Yaskawa INFORM job: X2_242(90,180)_HARDOX.JBI

/JOB
//NAME X2_242(90,180)_HARDOX
///FOLDERNAME X2
//POS
///NPOS 237,237,237,7,0,0
///TOOL 0
///POSTYPE PULSE
///PULSE
C00000=2000,-130321,-133031,0,28968,0
C00001=117091,-130321,-133031,-2123,28968,3391
C00002=159919,-130321,-133031,-2123,28968,3391
C00003=159919,-130321,-133031,-2123,87939,3391
C00004=105022,-108859,-78959,31083,72176,68730
C00005=151007,-25092,-39063,12800,65605,-78235
C00006=132593,67036,12002,14068,96381,-18620
C00007=133669,66493,21901,13656,90017,-18991
C00008=134323,89636,48442,14320,95130,-18049
C00009=134323,89198,49863,14289,94064,-18173
C00010=134090,67791,24612,13544,88977,-18967
C00011=134777,68740,27409,13371,87669,-18883
C00012=134996,69719,28564,13316,87433,-18835
C00013=134996,70471,26931,13315,88788,-18690
C00014=132576,62954,16151,13952,91863,-19138
C00015=158058,56370,5063,6789,93126,12165
C00016=161492,61731,13256,13118,78465,26852
C00017=161219,65846,21027,13360,75906,26484
C00018=158063,89381,46849,19528,82253,27212
C00019=158063,88948,47996,19566,81373,27071
C00020=160512,68550,26920,13794,73840,26014
C00021=160268,69078,27542,13908,73773,25920
C00022=161163,66904,24770,13484,74201,26276
C00023=161204,69435,27921,13504,73574,26218
C00024=161316,71640,30535,13487,73093,26202
C00025=161111,67594,24408,13472,74770,26322
C00026=161490,61134,14077,13154,77673,26766
C00027=158729,69794,18853,21227,92144,29458
C00028=158729,68570,20268,21195,90741,29212
C00029=158729,67854,21249,21182,89832,29052
C00030=158729,67915,21161,21182,89912,29066
C00031=158610,71039,24862,21209,89312,28918
C00032=158848,70143,22197,21157,90358,29181
C00033=158120,85702,32683,3458,102317,26701
C00034=153945,88580,39496,3983,99787,25284
C00035=153945,88046,40183,3975,99091,25261
C00036=153945,88140,40056,3976,99218,25265
C00037=153885,91305,44058,3974,98389,25220
C00038=154130,89669,40557,3958,99689,25341
C00039=154130,94954,36450,4054,104920,76820
C00040=150047,102272,56341,4455,96659,75219
C00041=150047,101948,56923,4449,96135,75198
C00042=150047,101994,56837,4450,96211,75201
C00043=150046,99636,53775,4457,96882,75225
C00044=149918,101619,55030,4477,97134,75192
C00045=163127,101976,55494,2716,96470,79472
C00046=163127,101465,56376,2711,95666,79454
C00047=163366,101791,56673,2679,95642,79533
C00048=163587,98952,52988,2655,96443,79621
C00049=163442,100538,53640,2678,96859,79582
C00050=163442,102448,51349,2698,99248,79634
C00051=156757,38630,-9639,10383,82653,33075
C00052=156267,40068,-956,10702,78181,32538
C00053=156202,41728,2024,10748,77230,32436
C00054=163721,62554,19620,-6039,89611,33850
C00055=164282,59884,16504,-9953,92188,36631
C00056=164282,59884,16504,-9953,92188,36631
C00057=161742,51287,7536,-7341,91343,24128
C00058=156677,44449,939,-1074,88896,15278
C00059=151279,46028,2666,6981,89616,6367
C00060=145657,58249,16160,8496,88116,4486
C00061=145657,58203,16260,8496,88033,4481
C00062=140244,72543,32903,17213,90923,-7444
C00063=141352,99915,64025,12711,93620,-30883
C00064=141512,101221,65699,12689,93243,-30868
C00065=122713,94046,59869,28177,93377,-67521
C00066=121487,97083,60557,28349,94790,-67637
C00067=133468,48615,1742,18804,93124,-11842
C00068=157997,71741,26694,3661,70569,66185
C00069=156653,80960,41725,4466,66130,65572
C00070=160707,58811,27097,-7838,50776,65613
C00071=161862,58527,28132,-10661,48808,66136
C00072=162060,71887,38599,-9565,55625,66013
C00073=162634,67727,36532,-11016,51381,65293
C00074=160821,61019,33044,-3636,43624,62105
C00075=154148,75334,40185,14517,57905,63097
C00076=154196,71820,32295,14055,60854,63507
C00077=153288,55034,31796,23088,50010,69293
C00078=151031,57353,45940,40148,40347,64995
C00079=150621,58129,46816,40537,40429,64769
C00080=149751,55668,48450,47014,34319,61006
C00081=150747,54467,47461,43008,31230,60446
C00082=154056,49858,42858,29251,25609,68749
C00083=154872,47959,37614,21306,28921,70888
C00084=159207,48403,28271,1768,40383,74494
C00085=149846,52946,33243,13952,46682,81563
C00086=149940,61587,46564,14806,43022,81015
C00087=146336,59430,51340,33146,36492,77110
C00088=145282,69746,63346,35645,35179,75711
C00089=143319,74757,70706,41882,34093,73425
C00090=141946,81470,79320,45365,33350,71705
C00091=140704,87470,87386,49528,32633,69847
C00092=140891,72507,62697,35215,38758,74780
C00093=145179,75875,59784,18821,43244,78638
C00094=142934,45174,24760,18717,49242,78806
C00095=150095,53682,32510,-1332,53765,80932
C00096=152813,60489,40795,-8113,54705,81636
C00097=150873,66241,46089,-11694,57678,80313
C00098=150873,66241,46089,-11694,57678,80313
C00099=147508,105073,69525,-3796,81278,78133
C00100=142743,125321,87945,7862,87558,77766
C00101=142103,130944,97278,17055,86189,78095
C00102=142103,130944,97278,17055,86189,78095
C00103=140795,85514,43044,21761,79618,77170
C00104=152813,60488,40794,-8113,54705,81636
C00105=153944,68685,21473,-9620,73495,76932
C00106=130978,99619,55052,27897,98813,81953
C00107=131949,98702,57308,26564,98678,82113
C00108=135763,95134,52790,26294,98361,83439
C00109=135763,95134,52790,26294,98361,83439
C00110=137181,56813,10142,24264,84548,80887
C00111=143258,42401,-4436,10530,76127,78768
C00112=143836,46028,-2345,1916,78517,77139
C00113=143836,46027,-2345,1916,78517,77139
C00114=145204,85743,36053,-2217,97184,77304
C00115=136098,105638,63245,17527,100626,82759
C00116=136098,107050,60359,17719,103015,83112
C00117=136992,102223,50247,17761,104726,73980
C00118=140383,74909,23622,16817,99949,37801
C00119=151007,-25092,-39063,12800,65605,-78235
C00120=105022,-108859,-78959,31083,72176,68730
C00121=159919,-130321,-133031,-2123,87939,3391
C00122=159919,-130321,-133031,-2123,28968,3391
C00123=117091,-130321,-133031,-2123,28968,3391
C00124=-31465,-130321,-133031,-2123,28968,3391
C00125=-31465,-130321,-133031,-2123,28968,3391
C00126=-70388,-93367,-87979,-22259,92531,40632
C00127=-132234,14944,-6259,-12342,59781,23208
C00128=-146205,63473,16177,-10072,90044,15024
C00129=-148576,68007,22640,-9405,88157,14412
C00130=-146386,94591,54398,-14629,94983,13774
C00131=-146332,95037,56689,-14603,93850,13927
C00132=-148776,67777,25971,-9352,86001,14507
C00133=-149047,69084,27509,-9276,85699,14442
C00134=-148423,68574,25700,-9447,86607,14574
C00135=-146195,62986,16971,-10071,89317,15086
C00136=-176137,58081,9771,3198,80109,-33161
C00137=-174052,65626,21441,2357,76742,-32574
C00138=-170116,81131,36386,-5185,84146,-32467
C00139=-170116,80866,36882,-5187,83709,-32446
C00140=-173210,63680,20711,2005,76169,-32311
C00141=-172556,64401,21545,1729,76012,-32099
C00142=-173019,62971,18478,1917,77173,-32231
C00143=-167045,54371,14180,-12829,67421,-32117
C00144=-167300,57261,17419,-12739,66888,-32149
C00145=-166775,56105,16119,-12998,67167,-31995
C00146=-174959,61653,15361,2721,78467,-32830
C00147=-175740,53447,3523,-48,85497,-33645
C00148=-175360,51508,3913,-186,84262,-33527
C00149=-175360,51073,4489,-186,83684,-33526
C00150=-175360,51149,4385,-186,83787,-33526
C00151=-175249,53641,7148,-228,83367,-33490
C00152=-175337,53338,6811,-195,83419,-33517
C00153=-175826,53926,7466,-13,83318,-33670
C00154=-175473,53555,5734,-142,84193,-33561
C00155=-144289,28411,-23210,-11283,91029,-24419
C00156=-143356,27785,-20851,-11589,89401,-23986
C00157=-143356,27161,-20168,-11587,88676,-23918
C00158=-143356,27239,-20255,-11587,88767,-23927
C00159=-143527,29595,-17924,-11529,88526,-23958
C00160=-143558,29339,-18180,-11519,88548,-23971
C00161=-144383,29127,-18388,-11237,88464,-24218
C00162=-144124,29609,-19345,-11326,89318,-24216
C00163=-152231,56674,-9545,3171,107413,-78802
C00164=-144736,71330,18445,-1025,104772,-77201
C00165=-144312,71202,19502,-1074,104058,-77059
C00166=-144312,70917,19790,-1073,103735,-77057
C00167=-144312,71001,19706,-1073,103831,-77057
C00168=-144182,68430,16646,-1091,104394,-77022
C00169=-145749,70587,16703,-901,105452,-77530
C00170=-159632,68614,11640,838,107552,-81931
C00171=-159546,67950,14693,818,105331,-81920
C00172=-159546,67280,15309,815,104608,-81925
C00173=-159546,67371,15221,815,104708,-81925
C00174=-159612,64750,12141,826,105257,-81943
C00175=-159714,67342,13242,842,105910,-81972
C00176=-155595,63448,7116,-8240,93528,-47643
C00177=-153862,58220,7137,-12336,84382,-31788
C00178=-154888,58914,9595,-11964,83110,-31986
C00179=-146509,53782,12657,-29932,73803,-35700
C00180=-161952,90743,44124,6697,92827,-37840
C00181=-160577,82650,33986,6445,94790,-37296
C00182=-160577,82650,33986,6445,94790,-37296
C00183=-159985,80927,31860,6330,95170,-37090
C00184=-155420,72888,22340,-1514,95229,-24069
C00185=-153394,77654,27323,-2558,97409,-16743
C00186=-148113,87914,39576,-10194,100615,205
C00187=-139080,92738,49536,-22064,95192,5031
C00188=-139986,94005,50057,-15877,93351,16845
C00189=-139980,94102,50182,-15876,93326,16850
C00190=-138241,102836,62169,-17611,90107,30313
C00191=-138415,104761,64681,-17573,89538,30337
C00192=-138485,105412,65534,-17560,89343,30340
C00193=-137728,105908,62856,-17713,91318,30315
C00194=-129809,68648,23314,-23742,79294,62187
C00195=-130521,38108,-11366,-22924,75116,53839
C00196=-144715,56131,10361,-11744,72134,-27543
C00197=-151566,59831,28742,2859,46138,-64220
C00198=-152051,66360,37815,3410,43933,-64521
C00199=-152374,66785,38353,3707,43835,-64678
C00200=-153165,73631,47658,1794,40169,-65578
C00201=-151811,68486,39030,-4846,43626,-66812
C00202=-148976,61300,30711,-7226,45253,-65595
C00203=-146833,59843,35175,-15333,37075,-63759
C00204=-143542,60593,37879,-27310,36429,-62771
C00205=-141155,67086,46027,-31931,35473,-60937
C00206=-143111,63918,40413,-22730,36091,-62179
C00207=-143710,65185,41996,-20330,35825,-62036
C00208=-139198,78346,59128,-30813,32871,-58285
C00209=-141383,82478,55565,-14874,41935,-61497
C00210=-145119,87922,62530,-17293,47365,-79425
C00211=-155100,67864,30953,12017,66106,-80987
C00212=-154047,73145,41863,11861,62043,-81030
C00213=-149809,72408,41128,9597,61562,-79468
C00214=-149809,72408,41128,9597,61562,-79468
C00215=-147962,104367,73434,5634,72990,-78503
C00216=-142842,140662,110237,-7498,79163,-77196
C00217=-145202,120199,82006,-7395,87027,-78490
C00218=-145202,120199,82006,-7395,87027,-78490
C00219=-142893,79503,35750,-14031,77749,-76980
C00220=-154047,73145,41863,11861,62043,-81030
C00221=-154847,69851,34699,12006,64817,-81032
C00222=-149316,91814,55261,-16182,79418,-82240
C00223=-150157,103206,68826,-20327,87511,-84213
C00224=-150410,102909,71857,-20845,86766,-84223
C00225=-154299,103919,73243,-20299,85488,-85396
C00226=-154299,103919,73243,-20299,85488,-85396
C00227=-159714,64678,27666,-9684,74240,-84843
C00228=-166555,65945,28804,6708,73710,-85034
C00229=-165808,57994,22044,12876,71037,-84145
C00230=-165808,57994,22044,12876,71037,-84145
C00231=-165613,93091,57596,12794,85266,-82832
C00232=-150410,102909,71857,-20845,86766,-84223
C00233=-150622,105536,71839,-20808,87992,-84510
C00234=-140496,9250,-2578,-20724,48099,-77689
C00235=-103999,-84119,-66645,-26288,35960,-55555
C00236=2000,-130321,-133031,0,28968,0
BC00000=147988,698532,1075229
BC00001=188414,1188203,1075229
BC00002=367660,1354304,1075229
BC00003=367660,1362196,1075229
BC00004=367660,1369205,239425
BC00005=367660,1369205,202835
BC00006=311811,1355257,45063
BC00007=311811,1355257,45063
BC00008=311811,1355257,45063
BC00009=311811,1355257,45063
BC00010=311811,1355257,45063
BC00011=311811,1355257,45063
BC00012=311811,1355257,45063
BC00013=311811,1355257,45063
BC00014=311811,1355257,45063
BC00015=362430,1330918,31815
BC00016=380287,1344786,8254
BC00017=380287,1344786,8254
BC00018=380287,1344786,8254
BC00019=380287,1344786,8254
BC00020=380287,1344786,8254
BC00021=380287,1344786,8254
BC00022=380287,1344786,8254
BC00023=380287,1344786,8254
BC00024=380287,1344786,8254
BC00025=380287,1344786,8254
BC00026=380287,1344786,8254
BC00027=380287,1344786,8254
BC00028=380287,1344786,8254
BC00029=380287,1344786,8254
BC00030=380287,1344786,8254
BC00031=380287,1344786,8254
BC00032=380287,1344786,8254
BC00033=380287,1344786,8254
BC00034=380287,1344786,8254
BC00035=380287,1344786,8254
BC00036=380287,1344786,8254
BC00037=380287,1344786,8254
BC00038=380287,1344786,8254
BC00039=380287,1344786,8254
BC00040=380287,1344786,8254
BC00041=380287,1344786,8254
BC00042=380287,1344786,8254
BC00043=380287,1344786,8254
BC00044=380287,1344786,8254
BC00045=380287,1344786,8254
BC00046=380287,1344786,8254
BC00047=380287,1344786,8254
BC00048=380287,1344786,8254
BC00049=380287,1344786,8254
BC00050=380287,1344786,8254
BC00051=343088,1328821,53324
BC00052=343088,1328821,53324
BC00053=343089,1328822,53323
BC00054=343088,1328821,53324
BC00055=343088,1328822,53323
BC00056=343088,1328822,53323
BC00057=343088,1328821,53324
BC00058=343088,1328821,53321
BC00059=343088,1328821,53322
BC00060=343088,1328821,53322
BC00061=343088,1328821,53322
BC00062=343088,1328821,53322
BC00063=343088,1328821,53322
BC00064=343088,1328821,53322
BC00065=294664,1328821,53324
BC00066=294664,1328821,53324
BC00067=320438,1350876,40928
BC00068=369061,1366246,27049
BC00069=367921,1368726,27049
BC00070=367921,1369019,27049
BC00071=367921,1369019,27049
BC00072=367921,1370068,27049
BC00073=367921,1370124,27049
BC00074=367921,1369271,27049
BC00075=367921,1369146,27049
BC00076=367921,1368921,27049
BC00077=384338,1356637,125684
BC00078=384338,1356637,125684
BC00079=384338,1356637,125684
BC00080=384338,1356637,125684
BC00081=384338,1356637,125684
BC00082=384338,1356637,125684
BC00083=384338,1356637,125684
BC00084=384338,1356637,125684
BC00085=367660,1358625,156647
BC00086=367660,1362300,156647
BC00087=367660,1361430,156647
BC00088=367660,1369205,156647
BC00089=367660,1369205,156647
BC00090=367660,1369205,156647
BC00091=367660,1369205,156647
BC00092=367660,1369205,156647
BC00093=367660,1369205,156647
BC00094=367660,1369205,156647
BC00095=367660,1369205,156647
BC00096=367660,1369205,156647
BC00097=367660,1369205,156647
BC00098=367660,1369205,156647
BC00099=367660,1369205,52075
BC00100=367660,1369205,3791
BC00101=367660,1369205,3791
BC00102=367660,1369205,3791
BC00103=367660,1369205,3791
BC00104=367660,1369205,156647
BC00105=367660,1369205,3791
BC00106=306487,1369247,3106
BC00107=306487,1369247,3106
BC00108=306487,1369247,3106
BC00109=306487,1369247,3106
BC00110=306487,1369247,3106
BC00111=306487,1369247,3106
BC00112=306487,1369247,3106
BC00113=306487,1369247,3106
BC00114=306487,1369247,3106
BC00115=306487,1369247,3106
BC00116=306487,1369247,3106
BC00117=310172,1369244,15137
BC00118=324080,1369237,60547
BC00119=367660,1369205,202835
BC00120=367660,1369205,239425
BC00121=367660,1369205,1075229
BC00122=367660,1369205,1075229
BC00123=188414,1188203,1075229
BC00124=341076,698532,1075229
BC00125=341076,698532,1075229
BC00126=259006,668063,241967
BC00127=356776,668063,241967
BC00128=356776,780350,42923
BC00129=356776,780350,42923
BC00130=356776,780350,42923
BC00131=356776,780350,42923
BC00132=356776,780350,42923
BC00133=356776,780350,42923
BC00134=356776,780350,42923
BC00135=356776,780350,42923
BC00136=398174,798504,17447
BC00137=398174,798504,17447
BC00138=398174,798504,17447
BC00139=398174,798504,17447
BC00140=398174,798504,17447
BC00141=398174,798504,17447
BC00142=398174,798504,17447
BC00143=398174,798504,17447
BC00144=398174,798504,17447
BC00145=398174,798504,17447
BC00146=398174,798504,17447
BC00147=398174,798504,17447
BC00148=398174,798504,17447
BC00149=398174,798504,17447
BC00150=398174,798504,17447
BC00151=398174,798504,17447
BC00152=398174,798504,17447
BC00153=398174,798504,17447
BC00154=398174,798504,17447
BC00155=346534,799135,17447
BC00156=346534,799135,17447
BC00157=346534,799135,17447
BC00158=346534,799135,17447
BC00159=346534,799135,17447
BC00160=346534,799135,17447
BC00161=346534,799135,17447
BC00162=346534,799135,17447
BC00163=346534,799135,17447
BC00164=346534,799135,17447
BC00165=346534,799135,17447
BC00166=346534,799135,17447
BC00167=346534,799135,17447
BC00168=346534,799135,17447
BC00169=346534,799135,17447
BC00170=346534,799135,17447
BC00171=346534,799135,17447
BC00172=346534,799135,17447
BC00173=346534,799135,17447
BC00174=346534,799135,17447
BC00175=346534,799135,17447
BC00176=344927,786208,5513
BC00177=344192,780294,53
BC00178=344192,780294,53
BC00179=344192,780294,53
BC00180=344192,780294,53
BC00181=344192,780294,53
BC00182=344192,780294,53
BC00183=344192,780294,53
BC00184=344192,780294,51
BC00185=344192,780294,53
BC00186=344192,780294,53
BC00187=344192,780294,48
BC00188=344192,780294,48
BC00189=344192,780294,48
BC00190=344192,780294,48
BC00191=344192,780294,48
BC00192=344192,780294,48
BC00193=344192,780294,48
BC00194=326520,780294,53
BC00195=326520,780294,53
BC00196=339286,748170,17050
BC00197=345010,733770,24669
BC00198=345010,733770,24669
BC00199=345010,733770,24669
BC00200=345010,733770,24669
BC00201=345010,733770,24667
BC00202=345010,733770,24667
BC00203=345010,733770,24667
BC00204=345010,733770,24667
BC00205=345010,733770,24667
BC00206=345010,733770,24667
BC00207=345010,733770,24667
BC00208=345010,733770,24667
BC00209=345010,733770,24667
BC00210=372205,746718,70819
BC00211=372205,746718,70819
BC00212=372205,746718,70819
BC00213=372205,746718,70819
BC00214=372205,746718,70819
BC00215=372205,746718,70819
BC00216=372205,746718,7590
BC00217=364929,753663,7590
BC00218=364929,753663,7590
BC00219=364929,753663,7590
BC00220=372205,746718,70819
BC00221=372205,746718,70819
BC00222=372205,767322,70819
BC00223=372205,767322,70819
BC00224=372205,767322,70819
BC00225=372205,767322,70819
BC00226=372205,767322,70819
BC00227=372205,767322,70819
BC00228=372205,767322,70819
BC00229=372205,767323,70818
BC00230=372205,767323,70818
BC00231=372205,767323,70818
BC00232=372205,767322,70819
BC00233=372205,767322,70819
BC00234=372204,667822,309341
BC00235=335743,674329,471628
BC00236=200134,698532,1075229
EC00000=798156,1112951
EC00001=798156,1112951
EC00002=798156,1112951
EC00003=798156,1112951
EC00004=798156,1112951
EC00005=798156,1112951
EC00006=798156,1112951
EC00007=798156,1112951
EC00008=798156,1112951
EC00009=798156,1112951
EC00010=798156,1112951
EC00011=798156,1112951
EC00012=798156,1112951
EC00013=798156,1112951
EC00014=798156,1112951
EC00015=798156,1112951
EC00016=798156,1112951
EC00017=798156,1112951
EC00018=798156,1112951
EC00019=798156,1112951
EC00020=798156,1112951
EC00021=798156,1112951
EC00022=798156,1112951
EC00023=798156,1112951
EC00024=798156,1112951
EC00025=798156,1112951
EC00026=798156,1112951
EC00027=798156,1112951
EC00028=798156,1112951
EC00029=798156,1112951
EC00030=798156,1112951
EC00031=798156,1112951
EC00032=798156,1112951
EC00033=798156,1112951
EC00034=798156,1112951
EC00035=798156,1112951
EC00036=798156,1112951
EC00037=798156,1112951
EC00038=798156,1112951
EC00039=798156,1112951
EC00040=798156,1112951
EC00041=798156,1112951
EC00042=798156,1112951
EC00043=798156,1112951
EC00044=798156,1112951
EC00045=798156,1112951
EC00046=798156,1112951
EC00047=798156,1112951
EC00048=798156,1112951
EC00049=798156,1112951
EC00050=798156,1112951
EC00051=798156,1112951
EC00052=798156,1112951
EC00053=798155,1112949
EC00054=798156,1112951
EC00055=798155,1112950
EC00056=798155,1112950
EC00057=798156,1112951
EC00058=798154,1112949
EC00059=798155,1112950
EC00060=798155,1112950
EC00061=798155,1112950
EC00062=798155,1112950
EC00063=798155,1112950
EC00064=798155,1112950
EC00065=798156,1112951
EC00066=798156,1112951
EC00067=798156,1112951
EC00068=798156,1112951
EC00069=798156,1112951
EC00070=798156,1112951
EC00071=798156,1112951
EC00072=798156,1112951
EC00073=798156,1112951
EC00074=798156,1112951
EC00075=798156,1112951
EC00076=798156,1112951
EC00077=798156,1112951
EC00078=798156,1112951
EC00079=798156,1112951
EC00080=798156,1112951
EC00081=798156,1112951
EC00082=798156,1112951
EC00083=798156,1112951
EC00084=798156,1112951
EC00085=798156,1112951
EC00086=798156,1112951
EC00087=798156,1112951
EC00088=798156,1112951
EC00089=798156,1112951
EC00090=798156,1112951
EC00091=798156,1112951
EC00092=798156,1112951
EC00093=798156,1112951
EC00094=798156,1112951
EC00095=798156,1112951
EC00096=798156,1112951
EC00097=798156,1112951
EC00098=798156,1112951
EC00099=798156,1112951
EC00100=798156,1112951
EC00101=798156,1112951
EC00102=798156,1112951
EC00103=798156,1112951
EC00104=798156,1112951
EC00105=798156,1112951
EC00106=798156,1112951
EC00107=798156,1112951
EC00108=798156,1112951
EC00109=798156,1112951
EC00110=798156,1112951
EC00111=798156,1112951
EC00112=798156,1112951
EC00113=798156,1112951
EC00114=798156,1112951
EC00115=798156,1112951
EC00116=798156,1112951
EC00117=798156,1112951
EC00118=798155,1112950
EC00119=798156,1112951
EC00120=798156,1112951
EC00121=798156,1112951
EC00122=798156,1112951
EC00123=798156,1112951
EC00124=798156,1112951
EC00125=-798156,1112951
EC00126=-798156,1112951
EC00127=-798156,1112951
EC00128=-798156,1112951
EC00129=-798156,1112951
EC00130=-798156,1112951
EC00131=-798156,1112951
EC00132=-798156,1112951
EC00133=-798156,1112951
EC00134=-798156,1112951
EC00135=-798156,1112951
EC00136=-798156,1112951
EC00137=-798156,1112951
EC00138=-798156,1112951
EC00139=-798156,1112951
EC00140=-798156,1112951
EC00141=-798156,1112951
EC00142=-798156,1112951
EC00143=-798156,1112951
EC00144=-798156,1112951
EC00145=-798156,1112951
EC00146=-798156,1112951
EC00147=-798156,1112951
EC00148=-798156,1112951
EC00149=-798156,1112951
EC00150=-798156,1112951
EC00151=-798156,1112951
EC00152=-798156,1112951
EC00153=-798156,1112951
EC00154=-798156,1112951
EC00155=-798156,1112951
EC00156=-798156,1112951
EC00157=-798156,1112951
EC00158=-798156,1112951
EC00159=-798156,1112951
EC00160=-798156,1112951
EC00161=-798156,1112951
EC00162=-798156,1112951
EC00163=-798156,1112951
EC00164=-798156,1112951
EC00165=-798156,1112951
EC00166=-798156,1112951
EC00167=-798156,1112951
EC00168=-798156,1112951
EC00169=-798156,1112951
EC00170=-798156,1112951
EC00171=-798156,1112951
EC00172=-798156,1112951
EC00173=-798156,1112951
EC00174=-798156,1112951
EC00175=-798156,1112951
EC00176=-798156,1112951
EC00177=-798156,1112951
EC00178=-798156,1112951
EC00179=-798156,1112951
EC00180=-798156,1112951
EC00181=-798156,1112951
EC00182=-798156,1112951
EC00183=-798156,1112951
EC00184=-798155,1112951
EC00185=-798156,1112951
EC00186=-798156,1112951
EC00187=-798154,1112952
EC00188=-798154,1112952
EC00189=-798154,1112952
EC00190=-798154,1112952
EC00191=-798154,1112952
EC00192=-798154,1112952
EC00193=-798154,1112952
EC00194=-798156,1112951
EC00195=-798156,1112951
EC00196=-798156,1112951
EC00197=-798155,1112951
EC00198=-798155,1112951
EC00199=-798155,1112951
EC00200=-798155,1112951
EC00201=-798154,1112952
EC00202=-798154,1112952
EC00203=-798154,1112952
EC00204=-798154,1112952
EC00205=-798154,1112952
EC00206=-798154,1112952
EC00207=-798154,1112952
EC00208=-798154,1112952
EC00209=-798154,1112952
EC00210=-798156,1112951
EC00211=-798156,1112951
EC00212=-798156,1112951
EC00213=-798156,1112951
EC00214=-798156,1112951
EC00215=-798156,1112951
EC00216=-798156,1112951
EC00217=-798156,1112951
EC00218=-798156,1112951
EC00219=-798156,1112951
EC00220=-798156,1112951
EC00221=-798156,1112951
EC00222=-798156,1112951
EC00223=-798156,1112951
EC00224=-798156,1112951
EC00225=-798156,1112951
EC00226=-798156,1112951
EC00227=-798156,1112951
EC00228=-798156,1112951
EC00229=-798154,1112952
EC00230=-798154,1112952
EC00231=-798154,1112952
EC00232=-798156,1112951
EC00233=-798156,1112951
EC00234=-798155,1112951
EC00235=-798155,1112951
EC00236=-798156,1112951
///POSTYPE BASE
///RECTAN
///RCONF 0,0,0,0,0,0,0,0,0,0,0,0,0,0,0,0,0,0,0,0,0,0,0,0
P00006=0.222,-3.123,-1.508,0.0000,0.0000,0.0000
P00021=-0.225,-6.128,-0.405,0.0000,0.0000,0.0000
P00022=0.222,-3.123,-1.508,0.0000,0.0000,0.0000
P00031=1.853,-0.001,-1.549,0.0000,0.0000,0.0000
P00032=1.957,0.503,-7.217,0.0000,0.0000,0.0000
///RCONF 0,0,0,0,1,0,0,0,0,0,0,0,0,0,0,0,0,0,0,0,0,0,0,0
P00033=-0.123,0.612,-5.012,0.0000,0.0000,0.0000
///RCONF 0,0,0,0,0,0,0,0,0,0,0,0,0,0,0,0,0,0,0,0,0,0,0,0
P00034=-0.304,0.773,-2.693,0.0000,0.0000,0.0000
//INST
///DATE 2024/12/13 09:44
///ATTR SC,RW
///GROUP1 RB1,BS1
///GROUP2 ST1
NOP
'X2_242(90,180)
'-90,0
MOVJ C00000 BC00000 VJ=100.00  +MOVJ EC00000 VJ=100.00
MOVJ C00001 BC00001 VJ=80.00  +MOVJ EC00001 VJ=100.00
MOVJ C00002 BC00002 VJ=70.00  +MOVJ EC00002 VJ=100.00
MOVJ C00003 BC00003 VJ=100.00  +MOVJ EC00003 VJ=100.00
MOVJ C00004 BC00004 VJ=100.00  +MOVJ EC00004 VJ=100.00
MOVJ C00005 BC00005 VJ=100.00  +MOVJ EC00005 VJ=100.00
'Path S4220
SFTOF3D
MOVJ C00006 BC00006 VJ=100.00  +MOVJ EC00006 VJ=100.00
MOVL C00007 BC00007 V=666.7  +MOVJ EC00007 VJ=100.00
SMOVL C00008 BC00008 V=166.7  +MOVJ EC00008
SREFP 3 C00009 BC00009  +REFP EC00009
CALL JOB:SEARCH-R1-S13D
SET P022 P006
SFTON3D P022
SMOVL C00010 BC00010 V=166.7  +MOVJ EC00010
SMOVL C00011 BC00011 V=166.7  +MOVJ EC00011
SREFP 3 C00012 BC00012  +REFP EC00012
CALL JOB:SEARCH-R1-S13D
SET P022 P006
SFTON3D P022
SMOVL C00013 BC00013 V=166.7  +MOVJ EC00013
MOVL C00014 BC00014 V=1000.0  +MOVJ EC00014 VJ=100.00
'EndPath S4220
MOVJ C00015 BC00015 VJ=100.00  +MOVJ EC00015 VJ=100.00
'Path S3549
SFTOF3D
MOVJ C00016 BC00016 VJ=100.00  +MOVJ EC00016 VJ=100.00
MOVL C00017 BC00017 V=666.7  +MOVJ EC00017 VJ=100.00
SMOVL C00018 BC00018 V=166.7  +MOVJ EC00018
SREFP 3 C00019 BC00019  +REFP EC00019
CALL JOB:SEARCH-R1-S13D
SET P021 P006
SFTON3D P021
SMOVL C00020 BC00020 V=166.7  +MOVJ EC00020
SREFP 3 C00021 BC00021  +REFP EC00021
CALL JOB:SEARCH-R1-S13D
SET P021 P006
SFTON3D P021
SMOVL C00022 BC00022 V=166.7  +MOVJ EC00022
SMOVL C00023 BC00023 V=166.7  +MOVJ EC00023
SREFP 3 C00024 BC00024  +REFP EC00024
CALL JOB:SEARCH-R1-S13D
SET P021 P006
SFTON3D P021
SMOVL C00025 BC00025 V=166.7  +MOVJ EC00025
MOVL C00026 BC00026 V=1000.0  +MOVJ EC00026 VJ=100.00
'EndPath S3549
'Path W3550
SFTOF3D
SSFTOF
SMOVL C00027 BC00027 V=333.3  +MOVJ EC00027
SMOVL C00028 BC00028 V=333.3  +MOVJ EC00028
SREFP 3 C00029 BC00029  +REFP EC00029
CALL JOB:SEARCH-R1-S13D
SET P031 P006
SFTON3D P031
SMOVL C00030 BC00030 V=166.7  +MOVJ EC00030
SREFP 3 C00031 BC00031  +REFP EC00031
CALL JOB:SEARCH-R1-S13D
SET P031 P006
SFTON3D P031
SMOVL C00032 BC00032 V=166.7  +MOVJ EC00032
SFTOF3D
SMOVL C00033 BC00033 V=333.3  +MOVJ EC00033
SMOVL C00034 BC00034 V=333.3  +MOVJ EC00034
SREFP 3 C00035 BC00035  +REFP EC00035
CALL JOB:SEARCH-R1-S13D
SET P033 P006
SFTON3D P033
SMOVL C00036 BC00036 V=333.3  +MOVJ EC00036
SREFP 3 C00037 BC00037  +REFP EC00037
CALL JOB:SEARCH-R1-S13D
SET P033 P006
SFTON3D P033
SMOVL C00038 BC00038 V=333.3  +MOVJ EC00038
SFTOF3D
SMOVL C00039 BC00039 V=333.3  +MOVJ EC00039
SMOVL C00040 BC00040 V=333.3  +MOVJ EC00040
SREFP 3 C00041 BC00041  +REFP EC00041
CALL JOB:SEARCH-R1-S13D
SET P034 P006
SFTON3D P034
SMOVL C00042 BC00042 V=333.3  +MOVJ EC00042
SREFP 3 C00043 BC00043  +REFP EC00043
CALL JOB:SEARCH-R1-S13D
SET P034 P006
SFTON3D P034
SMOVL C00044 BC00044 V=333.3  +MOVJ EC00044
SFTOF3D
SMOVL C00045 BC00045 V=333.3  +MOVJ EC00045
SREFP 3 C00046 BC00046  +REFP EC00046
CALL JOB:SEARCH-R1-S13D
SET P032 P006
SFTON3D P032
SMOVL C00047 BC00047 V=333.3  +MOVJ EC00047
SREFP 3 C00048 BC00048  +REFP EC00048
CALL JOB:SEARCH-R1-S13D
SET P032 P006
SFTON3D P032
SMOVL C00049 BC00049 V=333.3  +MOVJ EC00049
SMOVL C00050 BC00050 V=333.3  +MOVJ EC00050
SFTOF3D
SFTON3D P021
MOVJ C00051 BC00051 VJ=100.00  +MOVJ EC00051 VJ=100.00
SMOVL C00052 BC00052 V=666.7  +MOVJ EC00052
SMOVL C00053 BC00053 V=166.7 PL=0  +MOVJ EC00053
MACRO1 MJ#(0) ARGF9
ARCON
SMOVL C00054 BC00054 V=8.3  +MOVJ EC00054
SMOVL C00055 BC00055 V=8.3  +MOVJ EC00055
SMOVC C00056 BC00056 V=10.0  +MOVJ EC00056
SMOVC C00057 BC00057 V=10.0  +MOVJ EC00057
SFTON3D P022
SMOVC C00058 BC00058 V=10.0  +MOVJ EC00058
SMOVC C00059 BC00059 V=10.0  +MOVJ EC00059
SMOVL C00060 BC00060 V=10.0  +MOVJ EC00060
SFTON3D P021
SMOVC C00061 BC00061 V=10.0  +MOVJ EC00061
SMOVC C00062 BC00062 V=10.0  +MOVJ EC00062
SMOVC C00063 BC00063 V=10.0  +MOVJ EC00063
SMOVC C00064 BC00064 V=8.3  +MOVJ EC00064
ARCOF
SMOVL C00065 BC00065 V=800.0  +MOVJ EC00065
SMOVL C00066 BC00066 V=1000.0  +MOVJ EC00066
SFTOF3D
'EndPath W3550
MOVJ C00067 BC00067 VJ=100.00  +MOVJ EC00067 VJ=100.00
'Path W3552
SFTOF3D
SFTON3D P021
MOVJ C00068 BC00068 VJ=100.00  +MOVJ EC00068 VJ=100.00
SMOVL C00069 BC00069 V=800.0  +MOVJ EC00069
SMOVL C00070 BC00070 V=166.7  +MOVJ EC00070
MACRO1 MJ#(0) ARGF21
ARCON
SMOVL C00071 BC00071 V=9.2  +MOVJ EC00071
SMOVL C00072 BC00072 V=9.2  +MOVJ EC00072
SMOVL C00073 BC00073 V=9.2  +MOVJ EC00073
SMOVL C00074 BC00074 V=9.2  +MOVJ EC00074
ARCOF
SMOVL C00075 BC00075 V=800.0  +MOVJ EC00075
SMOVL C00076 BC00076 V=1000.0  +MOVJ EC00076
SFTOF3D
'EndPath W3552
'Path W3553
SFTOF3D
SFTON3D P022
MOVJ C00077 BC00077 VJ=100.00  +MOVJ EC00077 VJ=100.00
SMOVL C00078 BC00078 V=166.7 PL=0  +MOVJ EC00078
ARCON
SMOVL C00079 BC00079 V=8.3  +MOVJ EC00079
SMOVL C00080 BC00080 V=8.3  +MOVJ EC00080
SMOVL C00081 BC00081 V=8.3  +MOVJ EC00081
SMOVL C00082 BC00082 V=8.3  +MOVJ EC00082
ARCOF
SMOVL C00083 BC00083 V=800.0  +MOVJ EC00083
SMOVL C00084 BC00084 V=1000.0  +MOVJ EC00084
SFTOF3D
'EndPath W3553
'Path W3554
SFTOF3D
SFTON3D P022
MOVJ C00085 BC00085 VJ=50.00  +MOVJ EC00085 VJ=100.00
SMOVL C00086 BC00086 V=500.0  +MOVJ EC00086
SMOVL C00087 BC00087 V=166.7 PL=0  +MOVJ EC00087
ARCON
SMOVL C00088 BC00088 V=8.3  +MOVJ EC00088
SMOVL C00089 BC00089 V=8.3  +MOVJ EC00089
SMOVL C00090 BC00090 V=8.3  +MOVJ EC00090
SMOVL C00091 BC00091 V=8.3  +MOVJ EC00091
ARCOF
SMOVL C00092 BC00092 V=800.0  +MOVJ EC00092
SMOVL C00093 BC00093 V=1000.0  +MOVJ EC00093
SFTOF3D
'EndPath W3554
SMOVL C00094 BC00094 V=333.3  +MOVJ EC00094
SFTON3D P033
SMOVL C00095 BC00095 V=333.3  +MOVJ EC00095
SMOVL C00096 BC00096 V=166.7 PL=0  +MOVJ EC00096
ARCON
SMOVL C00097 BC00097 V=10.0  +MOVJ EC00097
SMOVC C00098 BC00098 V=10.0  +MOVJ EC00098
SFTON3D P034
SMOVC C00099 BC00099 V=10.0  +MOVJ EC00099
SMOVC C00100 BC00100 V=10.0  +MOVJ EC00100
SFTON3D P033
SMOVL C00101 BC00101 V=10.0  +MOVJ EC00101
SMOVC C00102 BC00102 V=10.0  +MOVJ EC00102
SMOVC C00103 BC00103 V=11.7  +MOVJ EC00103
SMOVC C00104 BC00104 V=12.5  +MOVJ EC00104
ARCOF
SMOVL C00105 BC00105 V=333.3  +MOVJ EC00105
SFTOF3D
SFTON3D P032
SMOVL C00106 BC00106 V=333.3  +MOVJ EC00106
SMOVL C00107 BC00107 V=166.7 PL=0  +MOVJ EC00107
ARCON
SFTON3D P031
SMOVL C00108 BC00108 V=10.0  +MOVJ EC00108
SMOVC C00109 BC00109 V=10.0  +MOVJ EC00109
SMOVC C00110 BC00110 V=12.5  +MOVJ EC00110
SMOVC C00111 BC00111 V=12.5  +MOVJ EC00111
SFTON3D P032
SMOVL C00112 BC00112 V=10.0  +MOVJ EC00112
SMOVC C00113 BC00113 V=10.0  +MOVJ EC00113
SMOVC C00114 BC00114 V=12.5  +MOVJ EC00114
SMOVC C00115 BC00115 V=12.5  +MOVJ EC00115
ARCOF
SMOVL C00116 BC00116 V=333.3  +MOVJ EC00116
SFTOF3D
MOVJ C00117 BC00117 VJ=50.00  +MOVJ EC00117 VJ=0.78
MOVJ C00118 BC00118 VJ=50.00  +MOVJ EC00118 VJ=50.00
MOVJ C00119 BC00119 VJ=100.00  +MOVJ EC00119 VJ=100.00
MOVJ C00120 BC00120 VJ=100.00  +MOVJ EC00120 VJ=100.00
MOVJ C00121 BC00121 VJ=100.00  +MOVJ EC00121 VJ=100.00
MOVJ C00122 BC00122 VJ=100.00  +MOVJ EC00122 VJ=100.00
MOVJ C00123 BC00123 VJ=100.00  +MOVJ EC00123 VJ=100.00
MOVJ C00124 BC00124 VJ=100.00  +MOVJ EC00124 VJ=100.00
MOVJ C00125 BC00125 VJ=100.00  +MOVJ EC00125 VJ=100.00
'-90,180
CALL JOB:CLEAN-R1_KM_NEW
MOVJ C00126 BC00126 VJ=100.00  +MOVJ EC00126 VJ=100.00
MOVJ C00127 BC00127 VJ=100.00  +MOVJ EC00127 VJ=100.00
'Path S4222
SFTOF3D
MOVJ C00128 BC00128 VJ=100.00  +MOVJ EC00128 VJ=100.00
MOVL C00129 BC00129 V=666.7  +MOVJ EC00129 VJ=100.00
SMOVL C00130 BC00130 V=166.7  +MOVJ EC00130
SREFP 3 C00131 BC00131  +REFP EC00131
CALL JOB:SEARCH-R1-S13D
SET P022 P006
SFTON3D P022
SMOVL C00132 BC00132 V=166.7  +MOVJ EC00132
SREFP 3 C00133 BC00133  +REFP EC00133
CALL JOB:SEARCH-R1-S13D
SET P022 P006
SFTON3D P022
SMOVL C00134 BC00134 V=166.7  +MOVJ EC00134
SFTOF3D
MOVL C00135 BC00135 V=1000.0  +MOVJ EC00135 VJ=100.00
'EndPath S4222
'Path S4223
SFTOF3D
MOVJ C00136 BC00136 VJ=100.00  +MOVJ EC00136 VJ=100.00
MOVL C00137 BC00137 V=666.7  +MOVJ EC00137 VJ=100.00
SMOVL C00138 BC00138 V=166.7  +MOVJ EC00138
SREFP 3 C00139 BC00139  +REFP EC00139
CALL JOB:SEARCH-R1-S13D
SET P021 P006
SFTON3D P021
SMOVL C00140 BC00140 V=166.7  +MOVJ EC00140
SREFP 3 C00141 BC00141  +REFP EC00141
CALL JOB:SEARCH-R1-S13D
SET P021 P006
SFTON3D P021
SMOVL C00142 BC00142 V=166.7  +MOVJ EC00142
SMOVL C00143 BC00143 V=166.7  +MOVJ EC00143
SREFP 3 C00144 BC00144  +REFP EC00144
CALL JOB:SEARCH-R1-S13D
SET P021 P006
SFTON3D P021
SMOVL C00145 BC00145 V=166.7  +MOVJ EC00145
MOVL C00146 BC00146 V=1000.0  +MOVJ EC00146 VJ=100.00
SFTOF3D
MOVJ C00147 BC00147 VJ=50.00  +MOVJ EC00147 VJ=50.00
SMOVL C00148 BC00148 V=166.7  +MOVJ EC00148
SREFP 3 C00149 BC00149  +REFP EC00149
CALL JOB:SEARCH-R1-S13D
SET P031 P006
SFTON3D P031
SMOVL C00150 BC00150 V=166.7  +MOVJ EC00150
SREFP 3 C00151 BC00151  +REFP EC00151
CALL JOB:SEARCH-R1-S13D
SET P031 P006
SFTON3D P031
SMOVL C00152 BC00152 V=166.7  +MOVJ EC00152
SREFP 3 C00153 BC00153  +REFP EC00153
CALL JOB:SEARCH-R1-S13D
SET P031 P006
SFTON3D P031
SMOVL C00154 BC00154 V=166.7  +MOVJ EC00154
SFTOF3D
SMOVL C00155 BC00155 V=666.7  +MOVJ EC00155
SMOVL C00156 BC00156 V=166.7  +MOVJ EC00156
SREFP 3 C00157 BC00157  +REFP EC00157
CALL JOB:SEARCH-R1-S13D
SET P033 P006
SFTON3D P033
SMOVL C00158 BC00158 V=166.7  +MOVJ EC00158
SREFP 3 C00159 BC00159  +REFP EC00159
CALL JOB:SEARCH-R1-S13D
SET P033 P006
SFTON3D P033
SMOVL C00160 BC00160 V=166.7  +MOVJ EC00160
SREFP 3 C00161 BC00161  +REFP EC00161
CALL JOB:SEARCH-R1-S13D
SET P033 P006
SFTON3D P033
SMOVL C00162 BC00162 V=166.7  +MOVJ EC00162
SFTOF3D
SMOVL C00163 BC00163 V=666.7  +MOVJ EC00163
SMOVL C00164 BC00164 V=666.7  +MOVJ EC00164
SFTON3D P033
SMOVL C00165 BC00165 V=166.7  +MOVJ EC00165
SREFP 3 C00166 BC00166  +REFP EC00166
CALL JOB:SEARCH-R1-S13D
SET P034 P006
SFTON3D P034
SMOVL C00167 BC00167 V=166.7  +MOVJ EC00167
SREFP 3 C00168 BC00168  +REFP EC00168
CALL JOB:SEARCH-R1-S13D
SET P034 P006
SFTON3D P034
SMOVL C00169 BC00169 V=166.7  +MOVJ EC00169
SFTOF3D
SMOVL C00170 BC00170 V=666.7  +MOVJ EC00170
SFTON3D P031
SMOVL C00171 BC00171 V=166.7  +MOVJ EC00171
SREFP 3 C00172 BC00172  +REFP EC00172
CALL JOB:SEARCH-R1-S13D
SET P032 P006
SFTON3D P032
SMOVL C00173 BC00173 V=166.7  +MOVJ EC00173
SREFP 3 C00174 BC00174  +REFP EC00174
CALL JOB:SEARCH-R1-S13D
SET P032 P006
SFTON3D P032
SMOVL C00175 BC00175 V=166.7  +MOVJ EC00175
SFTOF3D
SFTOF3D
MOVJ C00176 BC00176 VJ=50.00  +MOVJ EC00176 VJ=50.00
MOVJ C00177 BC00177 VJ=100.00  +MOVJ EC00177 VJ=100.00
SFTON3D P021
MOVL C00178 BC00178 V=666.7  +MOVJ EC00178 VJ=100.00
SMOVL C00179 BC00179 V=166.7 PL=0  +MOVJ EC00179
MACRO1 MJ#(0) ARGF9
ARCON
SMOVL C00180 BC00180 V=10.0  +MOVJ EC00180
SMOVL C00181 BC00181 V=9.2  +MOVJ EC00181
SMOVC C00182 BC00182 V=10.0  +MOVJ EC00182
SMOVC C00183 BC00183 V=10.0  +MOVJ EC00183
SFTON3D P022
SMOVC C00184 BC00184 V=10.0  +MOVJ EC00184
SMOVC C00185 BC00185 V=10.0  +MOVJ EC00185
SMOVC C00186 BC00186 V=10.0  +MOVJ EC00186
SMOVL C00187 BC00187 V=10.0  +MOVJ EC00187
SMOVL C00188 BC00188 V=10.0  +MOVJ EC00188
SMOVC C00189 BC00189 V=9.2  +MOVJ EC00189
SFTON3D P021
SMOVC C00190 BC00190 V=10.0  +MOVJ EC00190
SMOVC C00191 BC00191 V=10.0  +MOVJ EC00191
SMOVL C00192 BC00192 V=10.0  +MOVJ EC00192
ARCOF
MOVL C00193 BC00193 V=800.0  +MOVJ EC00193 VJ=100.00
MOVL C00194 BC00194 V=1000.0  +MOVJ EC00194 VJ=100.00
'EndPath W4224
MOVJ C00195 BC00195 VJ=100.00  +MOVJ EC00195 VJ=100.00
MOVJ C00196 BC00196 VJ=100.00  +MOVJ EC00196 VJ=100.00
'Path W4225
SFTOF3D
SFTON3D P021
SMOVL C00197 BC00197 V=800.0  +MOVJ EC00197
SMOVL C00198 BC00198 V=166.7 PL=0  +MOVJ EC00198
MACRO1 MJ#(0) ARGF21
ARCON
SMOVL C00199 BC00199 V=7.5  +MOVJ EC00199
SMOVL C00200 BC00200 V=7.5  +MOVJ EC00200
ARCOF
SMOVL C00201 BC00201 V=800.0  +MOVJ EC00201
SMOVL C00202 BC00202 V=1000.0  +MOVJ EC00202
SFTOF3D
'EndPath W4225
'Path W4226
SFTOF3D
SFTON3D P022
SMOVL C00203 BC00203 V=166.7 PL=0  +MOVJ EC00203
ARCON
SMOVL C00204 BC00204 V=8.3  +MOVJ EC00204
SMOVL C00205 BC00205 V=8.3  +MOVJ EC00205
ARCOF
SMOVL C00206 BC00206 V=800.0  +MOVJ EC00206
SFTOF3D
'EndPath W4226
'Path W4227
SFTOF3D
SFTON3D P022
SMOVL C00207 BC00207 V=166.7 PL=0  +MOVJ EC00207
ARCON
SMOVL C00208 BC00208 V=7.5  +MOVJ EC00208
ARCOF
SMOVL C00209 BC00209 V=800.0  +MOVJ EC00209
SMOVL C00210 BC00210 V=1000.0  +MOVJ EC00210
SFTOF3D
'EndPath W4227
MOVL C00211 BC00211 V=666.7  +MOVJ EC00211 VJ=50.00
MACRO1 MJ#(0) ARGF9
SFTON3D P033
SMOVL C00212 BC00212 V=166.7 PL=0  +MOVJ EC00212
ARCON
SFTON3D P034
SMOVL C00213 BC00213 V=10.0  +MOVJ EC00213
SMOVC C00214 BC00214 V=13.3  +MOVJ EC00214
SMOVC C00215 BC00215 V=13.3  +MOVJ EC00215
SMOVC C00216 BC00216 V=13.3  +MOVJ EC00216
SFTON3D P033
SMOVL C00217 BC00217 V=10.0  +MOVJ EC00217
SMOVC C00218 BC00218 V=13.3  +MOVJ EC00218
SMOVC C00219 BC00219 V=13.3  +MOVJ EC00219
SMOVC C00220 BC00220 V=13.3  +MOVJ EC00220
ARCOF
SMOVL C00221 BC00221 V=333.3  +MOVJ EC00221
SFTOF3D
MOVL C00222 BC00222 V=333.3  +MOVJ EC00222 VJ=50.00
MOVL C00223 BC00223 V=333.3  +MOVJ EC00223 VJ=50.00
SFTON3D P032
SMOVL C00224 BC00224 V=166.7 PL=0  +MOVJ EC00224
ARCON
SFTON3D P031
SMOVL C00225 BC00225 V=10.0  +MOVJ EC00225
SMOVC C00226 BC00226 V=13.3  +MOVJ EC00226
SMOVC C00227 BC00227 V=13.3  +MOVJ EC00227
SMOVC C00228 BC00228 V=13.3  +MOVJ EC00228
SFTON3D P032
SMOVL C00229 BC00229 V=10.0  +MOVJ EC00229
SMOVC C00230 BC00230 V=13.3  +MOVJ EC00230
SMOVC C00231 BC00231 V=13.3  +MOVJ EC00231
SMOVC C00232 BC00232 V=13.3  +MOVJ EC00232
ARCOF
MOVL C00233 BC00233 V=333.3  +MOVJ EC00233 VJ=50.00
SFTOF3D
MOVJ C00234 BC00234 VJ=100.00  +MOVJ EC00234 VJ=100.00
MOVJ C00235 BC00235 VJ=100.00  +MOVJ EC00235 VJ=100.00
MOVJ C00236 BC00236 VJ=100.00  +MOVJ EC00236 VJ=100.00
END
